{attribute 'qualified_only'}

// Команди който идват от I&C

TYPE controlCommands :
(
	null		:= 0,
	stop,
	start
	
)DINT;
END_TYPE

(* stored: Version 1.1.0.1, ProductVersion 3.1.4024.3
   DUT controlCommands: Id {547dc515-945c-45fa-b4e7-0a730d22b29b} *)
